(* IEC 61131-3 sources: repolevel_ST_code_completion/output/0121完整版本/repoeval_Wrappers/readful_result_history, 1 file *)

(* ---- FB_Wrapper_0.st ---- *)
FUNCTION_BLOCK FB_Wrapper
VAR_INPUT
	in:BOOL;
END_VAR
VAR_OUTPUT
	out:BOOL;
END_VAR
VAR
	fb_teste: ARRAY [1..3] OF FB_Teste;
	index: INT;
END_VAR

fb_teste[1].SetTempo(delay := T#4S);
fb_teste[2].SetTempo(delay := T#1S);
fb_teste[3].SetTempo(delay := T#2S);

FOR index := 1 TO 3 DO
	IF in THEN
		fb_teste[index].mLiga();
	ELSE
		fb_teste[index].mDesliga();
	END_IF;
END_FOR;

FOR index := 1 TO 3 DO
	fb_teste[index].entrada := in;
	out := fb_teste[index].saida;
END_FOR;
END_FUNCTION_BLOCK
